FUNCTION_BLOCK CM_UnlockingPins EXTENDS CM_Base

VAR_INPUT
	i_stSettings : ST_SettingsUnlockingPins;
END_VAR

VAR
	// Control Modules
	s_cmValveUnlockingPinUpper : CM_ValveWithFB;
	s_cmValveUnlockingPinLower : CM_ValveWithFB;
	
	// Request
	s_bReqLock : BOOL;
	s_bReqUnlock : BOOL;
	
	// Status
	s_bStaIsLocked : BOOL;
	s_bStaIsUnlocked : BOOL;
	
	{attribute: 'Hide'}
	s_bStaPins : BOOL; //FALSE = Locked, TRUE = Unlocked
	
	// Alarms
	
	// Timers
END_VAR


SUPER^();

METHOD PROTECTED _m_Alarms : BOOL

IF NOT SUPER^._m_Alarms() THEN
	RETURN;
END_IF

s_bStaError := 
	s_cmValveUnlockingPinUpper.p_bStaError
	OR s_cmValveUnlockingPinLower.p_bStaError;

_m_Alarms := TRUE;
END_METHOD

METHOD PROTECTED _m_Devices : BOOL

IF NOT SUPER^._m_Devices() THEN
	RETURN;
END_IF

//Call lower-layer devices
s_cmValveUnlockingPinUpper(
	i_bReqEnable:= i_bReqEnable, 
	i_eCtrlMode:= i_eCtrlMode, 
	i_bCmdReset:= i_bCmdReset, 
	i_sCmName:= 'Upper Unlocking Pin');
	
s_cmValveUnlockingPinLower(
	i_bReqEnable:= i_bReqEnable, 
	i_eCtrlMode:= i_eCtrlMode, 
	i_bCmdReset:= i_bCmdReset, 
	i_sCmName:= 'Lower Unlocking Pin');	

//Control lower-layer devcies
IF s_bReqLock THEN
	s_cmValveUnlockingPinUpper.m_Off();
	s_cmValveUnlockingPinLower.m_Off();
ELSIF s_bReqUnlock THEN
	s_cmValveUnlockingPinUpper.m_On();
	s_cmValveUnlockingPinLower.m_On();
ELSE
	s_cmValveUnlockingPinUpper.m_Stop();
	s_cmValveUnlockingPinLower.m_Stop();
END_IF

//Statusses
s_bStaIsLocked := s_cmValveUnlockingPinUpper.p_bStaIsOff AND s_cmValveUnlockingPinLower.p_bStaIsOff;
s_bStaIsUnlocked := s_cmValveUnlockingPinUpper.p_bStaIsOn AND s_cmValveUnlockingPinLower.p_bStaIsOn;

s_bStaPins := NOT(s_bStaIsLocked) AND s_bStaIsUnlocked;

_m_Devices := TRUE;
END_METHOD

METHOD PROTECTED _m_Hmi : BOOL

IF NOT SUPER^._m_Hmi() THEN
	RETURN;
END_IF

_m_Hmi := TRUE;
END_METHOD

METHOD PROTECTED _m_Init : BOOL

IF NOT SUPER^._m_Init() THEN
	RETURN;
END_IF

s_cmValveUnlockingPinUpper.i_stSettings.tValveOffTimeout := i_stSettings.tPinsLockTimeout;
s_cmValveUnlockingPinUpper.i_stSettings.tValveOnTimeout := i_stSettings.tPinsUnlockTimeout;

s_cmValveUnlockingPinLower.i_stSettings.tValveOffTimeout := i_stSettings.tPinsLockTimeout;
s_cmValveUnlockingPinLower.i_stSettings.tValveOnTimeout := i_stSettings.tPinsUnlockTimeout;

_m_Init := TRUE;
END_METHOD

METHOD PROTECTED _m_Inputs : BOOL

IF NOT SUPER^._m_Inputs() THEN
	RETURN;
END_IF

_m_Inputs := TRUE;
END_METHOD

METHOD PROTECTED _m_Outputs : BOOL

IF NOT SUPER^._m_Outputs() THEN
	RETURN;
END_IF

_m_Outputs := TRUE;
END_METHOD

METHOD PUBLIC m_Lock : BOOL

IF NOT i_bReqEnable THEN 
	RETURN;
END_IF

s_bReqLock := TRUE;
s_bReqUnlock := FALSE;

m_Lock := TRUE;
END_METHOD

METHOD PUBLIC m_Stop : BOOL

IF NOT i_bReqEnable THEN 
	RETURN;
END_IF

s_bReqLock := FALSE;
s_bReqUnlock := FALSE;

m_Stop := TRUE;
END_METHOD

METHOD PUBLIC m_Unlock : BOOL

IF NOT i_bReqEnable THEN 
	RETURN;
END_IF

s_bReqLock := FALSE;
s_bReqUnlock := TRUE;

m_Unlock := TRUE;
END_METHOD

{attribute 'monitoring':='call'}
PROPERTY PUBLIC p_bStaIsLocked : BOOL
GET

p_bStaIsLocked := s_bStaIsLocked;
END_GET
END_PROPERTY

{attribute 'monitoring':='call'}
PROPERTY PUBLIC p_bStaIsUnlocked : BOOL
GET

p_bStaIsUnlocked := s_bStaIsUnlocked;
END_GET
END_PROPERTY

{attribute 'monitoring':='call'}
PROPERTY PUBLIC p_bStaPins : BOOL
GET

p_bStaPins := s_bStaPins;
END_GET
END_PROPERTY

END_FUNCTION_BLOCK

(* stored: Version 1.1.0.1, ProductVersion 3.1.4024.12
   POU CM_UnlockingPins: Id {5fe56a10-b71c-419b-b351-f5f486dbde09}, SpecialFunc None
   Folder Methods: Id {ac78ef67-937f-49b3-9f14-88c938c1bbfb}
   Folder Properties: Id {8bc233e1-01fd-4210-8ab8-ae64d186d63e}
   Method _m_Alarms: Id {ea5cad21-9a17-4158-8d08-1b5d16ae26f5}
   Method _m_Devices: Id {f60a6693-6f78-44cd-a431-f829a283907f}
   Method _m_Hmi: Id {77b901e0-422e-4a24-8e53-08b881d5ddf3}
   Method _m_Init: Id {93ef7758-cb22-4383-acb2-e5491d520152}
   Method _m_Inputs: Id {030cc6a8-1db9-4eae-8f1b-0418e1962d62}
   Method _m_Outputs: Id {d560a77e-4ac0-49ea-a274-79af6ce98b74}
   Method m_Lock: Id {e158fffe-3ba6-4cca-a58f-97d6d6a76dfd}
   Method m_Stop: Id {ef35ada3-3e61-44f8-a0db-52c7e98d97d4}
   Method m_Unlock: Id {78b5749d-bcc4-42c4-855c-1d5d73e418fd}
   Property p_bStaIsLocked: Id {282a8800-5642-4888-9825-fa627e6c8511}
   Get Get: Id {e7b862c3-96b3-46db-b4db-c270910db319}
   Property p_bStaIsUnlocked: Id {7b1c3043-cbbf-45f9-a2aa-422055fec057}
   Get Get: Id {5d0bde43-9a30-4fb6-bcea-5c2f62576ccd}
   Property p_bStaPins: Id {b88e9833-1584-424f-8640-cde12cd0eac1}
   Get Get: Id {be364070-1a7e-44e3-ad0a-6d99ee27e1f5} *)
